# B&R Automation Studio project SimPanel
Automation Studio 4.9

## Configuration Standard

### Task classes (Cpu.sw)
```
Cyclic#4:
  Aufgabe3 <- Aufgabe3.prg [disabled]
  Aufgabe4 <- Aufgabe4.prg [disabled]
  Aufgabe5 <- Aufgabe5.prg [disabled]
  Aufgabe6 <- Aufgabe6.prg [disabled]
  Aufgabe7 <- Aufgabe7.prg [disabled]
  Aufgabe8 <- Aufgabe8.prg
Binaries: udbdef, FWRules, TCData, sysconf, Role, User, iomap, ashwd, asfw, arconfig, ashwac
Libraries: standard
```

### Hardware
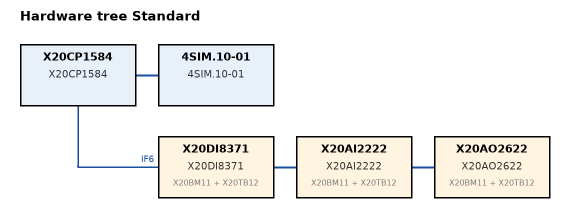
```
4SIM.10-01 : 4SIM.10-01 v1.3.0.0  [PLK1 -> X20CP1584.IF3 (NodeNumber=1) [Cable Type=PowerlinkCable, Length=10, Version=1.0.0.3]]
X20AI2222 : X20AI2222 v1.2.0.0  [SS1 -> X20TB12a.SS; SL -> X20BM11a.SL1]
X20AO2622 : X20AO2622 v1.3.0.0  [SS1 -> X20TB12b.SS; SL -> X20BM11b.SL1]
X20BM11 : X20BM11 v1.1.0.0  [X2X1 -> X20CP1584.IF6]
X20BM11a : X20BM11 v1.1.0.0  [X2X1 -> X20BM11.X2X2]
X20BM11b : X20BM11 v1.1.0.0  [X2X1 -> X20BM11a.X2X2]
X20CP1584 : X20CP1584 v1.10.0.0
  Connector IF2:
    ActivateDevice = 1
    Mode = Manual
    InternetAddress = 10.36.37.12
    SubnetMask = 255.255.255.0
  FileDevice1
  FileDeviceName1 = USER
  FileDevicePath1 = USER_PATH
X20DI8371 : X20DI8371 v1.4.0.0  [SS1 -> X20TB12.SS; SL -> X20BM11.SL1]
X20TB12 : X20TB12 v1.0.0.0
X20TB12a : X20TB12 v1.0.0.0
X20TB12b : X20TB12 v1.0.0.0
```

### IoMap.iom - X20CP1584/IoMap.iom
```iecst
VAR_CONFIG
	::Sw1 AT %IX."4SIM.10-01".DigitalInput01;
	::LED1 AT %QX."4SIM.10-01".DigitalOutput01;
	::Sw2 AT %IX."4SIM.10-01".DigitalInput02;
	::BtnArray[0].Btn AT %IX."4SIM.10-01".DigitalInput03;
	::BtnArray[1].Btn AT %IX."4SIM.10-01".DigitalInput04;
	::BtnArray[2].Btn AT %IX."4SIM.10-01".DigitalInput05;
	::BtnArray[3].Btn AT %IX."4SIM.10-01".DigitalInput06;
	::LED2 AT %QX."4SIM.10-01".DigitalOutput02;
	::BtnArray[0].LEDR AT %QX."4SIM.10-01".DigitalOutput03;
	::BtnArray[0].LEDY AT %QX."4SIM.10-01".DigitalOutput04;
	::BtnArray[0].LEDG AT %QX."4SIM.10-01".DigitalOutput05;
	::BtnArray[1].LEDR AT %QX."4SIM.10-01".DigitalOutput06;
	::BtnArray[1].LEDY AT %QX."4SIM.10-01".DigitalOutput07;
	::BtnArray[1].LEDG AT %QX."4SIM.10-01".DigitalOutput08;
	::BtnArray[2].LEDR AT %QX."4SIM.10-01".DigitalOutput09;
	::BtnArray[2].LEDY AT %QX."4SIM.10-01".DigitalOutput10;
	::BtnArray[2].LEDG AT %QX."4SIM.10-01".DigitalOutput11;
	::BtnArray[3].LEDR AT %QX."4SIM.10-01".DigitalOutput12;
	::BtnArray[3].LEDY AT %QX."4SIM.10-01".DigitalOutput13;
	::BtnArray[3].LEDG AT %QX."4SIM.10-01".DigitalOutput14;
	::DISP AT %QW."4SIM.10-01".AnalogOutput01;
	::P1 AT %IW."4SIM.10-01".AnalogInput01;
	::P2 AT %IW."4SIM.10-01".AnalogInput02;
	::Btn7 AT %IX."4SIM.10-01".DigitalInput07;
	::K1 AT %IW."4SIM.10-01".Encoder01;
END_VAR
```

## Logical view

### Global.typ - Global data types
```iecst
TYPE
	Button_t : 	STRUCT
		Btn : BOOL;
		Btn_Rise : R_TRIG;
		LEDG : BOOL;
		LEDY : BOOL;
		LEDR : BOOL;
		Btn_LongRise : R_TRIG;
		Btn_TOn : TON;
	END_STRUCT;
END_TYPE
```

### Global.var - Global variables
```iecst
VAR
	Sw1 : BOOL;
	Sw1_Rise : R_TRIG;
	Sw2 : BOOL;
	BtnArray : ARRAY[0..3] OF Button_t;
	Btn7 : BOOL;
	LED1 : BOOL;
	LED2 : BOOL;
	DISP : INT;
	P1 : INT;
	P2 : INT;
	K1 : UINT;
	BtnDelay : TIME;
	BtnTOn : ARRAY[0..3] OF TON;
	Btn3Cnt : USINT;
END_VAR
```

### Program Logical/Aufgabe3 (ANSIC)

#### Cyclic.c
```c
#include <bur/plctypes.h>

#ifdef _DEFAULT_INCLUDES
#include <AsDefault.h>
#endif

#define BTN_NUMBER 4

R_TRIG_typ set_R_TRIG(R_TRIG_typ Rset, BOOL CLK);

void toggleLED(int index);

void _CYCLIC ProgramCyclic(void)
{
	int cnt;

	// Dedect Rising Edge of Switch 1
	Sw1_Rise = set_R_TRIG(Sw1_Rise, Sw1);

	// Dedect Rising Edge of Buttons 3-6
	for (cnt = 0; cnt < BTN_NUMBER; cnt++)
	{
		BtnArray[cnt].Btn_Rise = set_R_TRIG(BtnArray[cnt].Btn_Rise, BtnArray[cnt].Btn);
	}

	// Switch 1 turned on -> all red LEDs on
	if (Sw1_Rise.Q)
	{
		for(cnt = 0; cnt < BTN_NUMBER; cnt++)
		{
			BtnArray[cnt].LEDR = 1;
		}
	}

	// Check for Button Press -> Toggle LED
	for (cnt = 0; cnt < BTN_NUMBER; cnt++)
	{
		if (Sw1 && BtnArray[cnt].Btn_Rise.Q)
		{
			toggleLED(cnt);
		}
	}

	if (Sw1) LED1 = 1;
	else
	{
		// Turn all LEDs off
		LED1 = 0;

		for (cnt = 0; cnt < BTN_NUMBER; cnt++)
		{
			BtnArray[cnt].LEDR = 0;
			BtnArray[cnt].LEDY = 0;
			BtnArray[cnt].LEDG = 0;
		}
	}
}

R_TRIG_typ set_R_TRIG(R_TRIG_typ Rset, BOOL CLK)
{
	Rset.CLK = CLK;
	R_TRIG(&Rset);
	return Rset;
}

void toggleLED(int index)
{
	BtnArray[index].LEDR = !BtnArray[index].LEDR;
	BtnArray[index].LEDG = !BtnArray[index].LEDG;
}
```

#### Init.c
```c
#include <bur/plctypes.h>

#ifdef _DEFAULT_INCLUDES
	#include <AsDefault.h>
#endif

#define BTN_NUMBER 4

void _INIT ProgramInit(void)
{
	// Set all outputs to Zero

	LED1 = 0;
	LED2 = 0;
	DISP = 0;

	int cnt;
	for (cnt = 0; cnt < BTN_NUMBER; cnt++)
	{
		BtnArray[cnt].LEDR = 0;
		BtnArray[cnt].LEDY = 0;
		BtnArray[cnt].LEDG = 0;
	}
}
```

### Program Logical/Aufgabe4 (ANSIC)

#### Cyclic.c
```c
#include <bur/plctypes.h>

#ifdef _DEFAULT_INCLUDES
	#include <AsDefault.h>
#endif

#define BTN_NUMBER 4

R_TRIG_typ set_R_TRIG(R_TRIG_typ Rset, BOOL CLK);
TON_typ set_TON(TON_typ Tset, BOOL IN);

void toggleLED(int index);

void _CYCLIC ProgramCyclic(void)
{
	int cnt;

	// Dedect Rising Edge of Switch 1
	Sw1_Rise = set_R_TRIG(Sw1_Rise, Sw1);

	// Dedect Delay and Rising Edge Button 3-6
	for (cnt = 0; cnt < BTN_NUMBER; cnt++)
	{
		BtnTOn[cnt] = set_TON(BtnTOn[cnt], BtnArray[cnt].Btn);
		BtnArray[cnt].Btn_Rise = set_R_TRIG(BtnArray[cnt].Btn_Rise, BtnTOn[cnt].Q);
	}

	// Check if any Button Rise is true
	for (cnt = 0; cnt < BTN_NUMBER; cnt++)
	{
		if (Sw1 && BtnArray[cnt].Btn_Rise.Q)
		{
			toggleLED(cnt);
		}
	}

	// Switch 1 turned on -> all red LEDs on
	if (Sw1_Rise.Q)
	{
		for(cnt = 0; cnt < BTN_NUMBER; cnt++)
		{
			BtnArray[cnt].LEDR = 1;
		}
	}

	if (Sw1) LED1 = 1;
	else
	{
		// Turn all LEDs off
		LED1 = 0;

		for (cnt = 0; cnt < BTN_NUMBER; cnt++)
		{
			BtnArray[cnt].LEDR = 0;
			BtnArray[cnt].LEDY = 0;
			BtnArray[cnt].LEDG = 0;
		}
	}
}

R_TRIG_typ set_R_TRIG(R_TRIG_typ Rset, BOOL CLK)
{
	Rset.CLK = CLK;
	R_TRIG(&Rset);
	return Rset;
}

TON_typ set_TON(TON_typ TONset, BOOL IN)
{
	TONset.IN = IN;
	TONset.PT = BtnDelay;
	TON(&TONset);
	return TONset;
}

void toggleLED(int index)
{
	BtnArray[index].LEDR = !BtnArray[index].LEDR;
	BtnArray[index].LEDG = !BtnArray[index].LEDG;
}
```

#### Exit.c
```c
#include <bur/plctypes.h>

#ifdef _DEFAULT_INCLUDES
	#include <AsDefault.h>
#endif

#define BTN_NUMBER 4

void _EXIT ProgramExit(void)
{
	// Set all outputs to Zero

	LED1 = 0;
	LED2 = 0;
	DISP = 0;

	int cnt;
	for (cnt = 0; cnt < BTN_NUMBER; cnt++)
	{
		BtnArray[cnt].LEDR = 0;
		BtnArray[cnt].LEDY = 0;
		BtnArray[cnt].LEDG = 0;
	}
}
```

#### Init.c
```c
#include <bur/plctypes.h>

#ifdef _DEFAULT_INCLUDES
	#include <AsDefault.h>
#endif

#define BTN_NUMBER 4

void _INIT ProgramInit(void)
{
	// Set Delay Time
	BtnDelay = 3000; // 3000ms = 3s

	// Set all outputs to Zero

	LED1 = 0;
	LED2 = 0;
	DISP = 0;

	int cnt;
	for (cnt = 0; cnt < BTN_NUMBER; cnt++)
	{
		BtnArray[cnt].LEDR = 0;
		BtnArray[cnt].LEDY = 0;
		BtnArray[cnt].LEDG = 0;
	}
}
```

### Program Logical/Aufgabe5 (ANSIC)

#### Cyclic.c
```c
#include <bur/plctypes.h>

#ifdef _DEFAULT_INCLUDES
	#include <AsDefault.h>
#endif

void _CYCLIC ProgramCyclic(void)
{
	if (Sw1)
	{
		LED1 = 1;
		DISP = P1 / 327; // Values Range [0, 32767] => [0, 100]
	}
	else
	{
		LED1 = 0;
		DISP = 0;
	}
}
```

#### Exit.c
```c
#include <bur/plctypes.h>

#ifdef _DEFAULT_INCLUDES
	#include <AsDefault.h>
#endif

#define BTN_NUMBER 4

void _EXIT ProgramExit(void)
{
	// Set all outputs to Zero

	LED1 = 0;
	LED2 = 0;
	DISP = 0;

	int cnt;
	for (cnt = 0; cnt < BTN_NUMBER; cnt++)
	{
		BtnArray[cnt].LEDR = 0;
		BtnArray[cnt].LEDY = 0;
		BtnArray[cnt].LEDG = 0;
	}
}
```

### Program Logical/Aufgabe6 (ANSIC)

#### Cyclic.c
```c
#include <bur/plctypes.h>

#ifdef _DEFAULT_INCLUDES
	#include <AsDefault.h>
#endif

#define BTN_NUMBER 4

R_TRIG_typ set_R_TRIG(R_TRIG_typ Rset, BOOL CLK);
INT P_Value_100(INT P);

void _CYCLIC ProgramCyclic(void)
{
	int cnt;

	for (cnt = 0; cnt < BTN_NUMBER; cnt++)
	{
		BtnArray[cnt].Btn_Rise = set_R_TRIG(BtnArray[cnt].Btn_Rise, BtnArray[cnt].Btn);
	}

	// Switch 1
	if (Sw1)
	{
		LED1 = 1;
		DISP = P_Value_100(P1);
	}
	else
	{
		LED1 = 0;
	}

	// Switch 2
	if (Sw2)
	{
		LED2 = 1;
		DISP = P_Value_100(P2);
	}
	else
	{
		LED2 = 0;
	}

	if (!Sw1 && !Sw2)
	{
		// Sum
		if (BtnArray[0].Btn_Rise.Q)
		{
			DISP = P_Value_100(P1) + P_Value_100(P2);
		}
		// Difference
		if (BtnArray[1].Btn_Rise.Q)
		{
			DISP = P_Value_100(P1) - P_Value_100(P2);
		}
		// Product
		if (BtnArray[2].Btn_Rise.Q)
		{
			DISP = P_Value_100(P1) * P_Value_100(P2);
		}
		// Quotient
		if (BtnArray[3].Btn_Rise.Q && P_Value_100(P2) != 0)
		{
			DISP = P_Value_100(P1) / P_Value_100(P2);
		}
	}
}

R_TRIG_typ set_R_TRIG(R_TRIG_typ Rset, BOOL CLK)
{
	Rset.CLK = CLK;
	R_TRIG(&Rset);
	return Rset;
}

INT P_Value_100(INT P)
{
	return P / 327; // Values Range [0, 32767] => [0, 100]
}
```

### Program Logical/Aufgabe7 (ANSIC)

#### Cyclic.c
```c
#include <bur/plctypes.h>

#ifdef _DEFAULT_INCLUDES
	#include <AsDefault.h>
#endif

#define DI3 	0
#define DELAY	500	// ms

TON_typ set_TON(TON_typ TONset, BOOL IN);

void _CYCLIC ProgramCyclic(void)
{
	if (Sw1)
	{
		LED1 = 1;

		BtnTOn[DI3].IN = 1;

		if (BtnTOn[DI3].Q)
		{
			BtnArray[DI3].LEDR = !BtnArray[DI3].LEDR;
			BtnTOn[DI3].IN = 0;
		}

		BtnTOn[DI3] = set_TON(BtnTOn[DI3], BtnTOn[DI3].IN);
	}
	else
	{
		LED1 = 0;
		BtnArray[DI3].LEDR = 0;
	}
}

TON_typ set_TON(TON_typ TONset, BOOL IN)
{
	TONset.IN = IN;
	TONset.PT = DELAY;
	TON(&TONset);
	return TONset;
}
```

#### Init.c
```c
#include <bur/plctypes.h>

#ifdef _DEFAULT_INCLUDES
	#include <AsDefault.h>
#endif

#define BTN_NUMBER 4

void _INIT ProgramInit(void)
{
	// Set all outputs to Zero

	LED1 = 0;
	LED2 = 0;
	DISP = 0;

	int cnt;
	for (cnt = 0; cnt < BTN_NUMBER; cnt++)
	{
		BtnArray[cnt].LEDR = 0;
		BtnArray[cnt].LEDY = 0;
		BtnArray[cnt].LEDG = 0;
	}
}
```

### Program Logical/Aufgabe8 (ANSIC)

#### Cyclic.c
```c
#include <bur/plctypes.h>

#ifdef _DEFAULT_INCLUDES
	#include <AsDefault.h>
#endif

#define BTN_NUMBER 	4
#define DELAY		1000 // ms

R_TRIG_typ set_R_TRIG(R_TRIG_typ Rset, BOOL CLK);
TON_typ set_TON(TON_typ Tset, BOOL IN);
void toggleLEDshort(int index);
void toggleLEDlong(int index);

void _CYCLIC ProgramCyclic(void)
{
	int cnt;

	// Dedect Rising Edge of Switch 1
	Sw1_Rise = set_R_TRIG(Sw1_Rise, Sw1);

	// Dedect Rising Edge of Buttons 3-6
	for (cnt = 0; cnt < BTN_NUMBER; cnt++)
	{
		// short Rising Edge
		BtnArray[cnt].Btn_Rise = set_R_TRIG(BtnArray[cnt].Btn_Rise, BtnArray[cnt].Btn);

		// long Rising Edge
		BtnArray[cnt].Btn_TOn = set_TON(BtnArray[cnt].Btn_TOn, BtnArray[cnt].Btn);
		BtnArray[cnt].Btn_LongRise = set_R_TRIG(BtnArray[cnt].Btn_LongRise, BtnArray[cnt].Btn_TOn.Q);
	}

	// Switch 1 turned on -> all yellow LEDs on
	if (Sw1_Rise.Q)
	{
		for(cnt = 0; cnt < BTN_NUMBER; cnt++)
		{
			BtnArray[cnt].LEDY = 1;
		}
	}

	// Check for short and long Button Press -> Toggle LED
	for (cnt = 0; cnt < BTN_NUMBER; cnt++)
	{
		if (Sw1 && BtnArray[cnt].Btn_Rise.Q)
		{
			toggleLEDshort(cnt);
		}
		if (Sw1 && BtnArray[cnt].Btn_LongRise.Q)
		{
			toggleLEDlong(cnt);
		}
	}

	if (Sw1) LED1 = 1;
	else
	{
		// Turn all LEDs off
		LED1 = 0;

		for (cnt = 0; cnt < BTN_NUMBER; cnt++)
		{
			BtnArray[cnt].LEDR = 0;
			BtnArray[cnt].LEDY = 0;
			BtnArray[cnt].LEDG = 0;
		}
	}
}

R_TRIG_typ set_R_TRIG(R_TRIG_typ Rset, BOOL CLK)
{
	Rset.CLK = CLK;
	R_TRIG(&Rset);
	return Rset;
}

TON_typ set_TON(TON_typ TONset, BOOL IN)
{
	TONset.IN = IN;
	TONset.PT = DELAY;
	TON(&TONset);
	return TONset;
}

void toggleLEDshort(int index)
{
	if (BtnArray[index].LEDY == 1)
	{
		BtnArray[index].LEDR = 0;
		BtnArray[index].LEDY = 0;
		BtnArray[index].LEDG = 1;
	}
	else
	{
		BtnArray[index].LEDR = 0;
		BtnArray[index].LEDY = 1;
		BtnArray[index].LEDG = 0;
	}
}

void toggleLEDlong(int index)
{
	BtnArray[index].LEDR = 1;
	BtnArray[index].LEDY = 0;
	BtnArray[index].LEDG = 0;
}
```

Listed in the project but not available here: Logical/Libraries
